FUNCTION_BLOCK FB_ComponentEX EXTENDS FB_Component
VAR_INPUT
END_VAR
VAR_OUTPUT
END_VAR
VAR
	bReturn: 		BOOL;
	bError:			BOOL;
	bAbort:			BOOL;
	bStop:			BOOL;
	bPause:			BOOL;
	bHold:			BOOL;
	bComplete:		BOOL;
	bInformation:	BOOL;
	bWarning:		BOOL;
END_VAR

METHOD PROTECTED M_Execute : BOOL
VAR_INPUT
END_VAR
CASE fbSequence.P_Number OF
	E_Sequence.Start:
		fbSequence.M_Await('Start', T#0S, T#0S, TRUE, bReturn, 10);
	
	10:
		fbSequence.M_Await('Step 10', T#0S, T#0S, TRUE, bReturn, 20);
		
	20:
		fbSequence.M_Await('Step 20', T#0S, T#0S, FALSE, bReturn, E_Sequence.Done);	
		
	E_Sequence.Done:
		fbSequence.M_Reset();
		M_Execute:= TRUE;
		
END_CASE

IF bAbort THEN
	bAbort:= FALSE;
	fbEvent.M_AddSTRING('1');
	fbEvent.M_AddSTRING('2');
	fbEvent.M_AddSTRING('3');
	fbEvent.M_Abort('First Error Abort %s %s %s', 6);
END_IF

IF bStop THEN
	bStop:= FALSE;
	fbEvent.M_AddSTRING('a');
	fbEvent.M_AddSTRING('b');
	fbEvent.M_AddSTRING('c');
	fbEvent.M_Stop('First Error Stop', 7);
END_IF

IF bError THEN
	fbEvent.M_Error('First Error', 8);
END_IF

IF bPause THEN
	fbEvent.M_Pause('First Pause', 9);
END_IF

IF bHold THEN
	fbEvent.M_Hold('First Hold', 10);
END_IF

IF bComplete THEN
	fbEvent.M_Complete('First Complete', 11);	
END_IF

IF bInformation THEN
	fbEvent.M_Information('Info', 12);	
END_IF

IF bWarning THEN
	fbEvent.M_Warning('Warning', 13);	
END_IF
END_METHOD

END_FUNCTION_BLOCK

(* stored: Version 1.1.0.1
   POU FB_ComponentEX: Id {67ecce00-b6ba-4016-865f-4a4dfdc94a76}, SpecialFunc None
   Method M_Execute: Id {bba4d435-5736-45bd-97fd-4ceab6f0d012} *)
